// TIA Portal V19 export
FUNCTION_BLOCK "Robot_Modbus"   // FB1, LAD
{ S7_Optimized_Access := 'TRUE' }
// V.0.1.1 - Updated UR robot array address
// V.0.1.0 - Created function block
// stored: MemoryReserve 100, SetENOAutomatically false
   VAR_INPUT
      Proces_Item : Bool;
      Place_Item_Conveyor : Bool;
      Place_Item_Storage : Bool;
      Scrap_Item : Bool;
      Speed_Transport : Int := 10;
      Speed_Grinding : Int := 10;
      Grinding_Coordinates : Bool;
      HMI_String : String;
   END_VAR
   VAR_OUTPUT
      Working : Bool;
      Done : Bool;
      Error : Bool;
      Reached_Coordinates : Bool;
   END_VAR
   VAR
      DISCONNECT : Bool;
      Address : TCON_IP_v4;
      Receive_Data : Int;
      Send_Data : Array[0..63] of Bool;
      Send_Coordinates : Array[0..2] of Int;
      Letter_A : Array[0..20] of "XYZ_Coordinates";
      Letter_Steps { S7_SetPoint := 'True'} : Int;
      Rising_edge : Bool;
      String_To_Letter_Array : Array[0..16] of Char;
      String_Length : Int;
      Currently_Processing : Int;
      Send_Letter_A : Bool;
      Send_Letter_B : Bool;
      Send_Letter_C : Bool;
      MB_Client_Mode : Int;
      MB_Client_Modbus_Address : Int;
      For_Loop_Counter : Int;
   END_VAR
   // Address.InterfaceId := 64;
   // Address.ID := 1;
   // Address.ConnectionType := 11;
   // Address.ActiveEstablished := TRUE;
   // Address.RemoteAddress.ADDR[1] := 192;
   // Address.RemoteAddress.ADDR[2] := 168;
   // Address.RemoteAddress.ADDR[3] := 1;
   // Address.RemoteAddress.ADDR[4] := 51;
   // Address.RemotePort := 502;
   // Address.LocalPort := 502;
   // Letter_A[0..1].X := 4;
   // Letter_A[2].X := 42;
   // Letter_A[3].X := 56;
   // Letter_A[4].X := 98;
   // Letter_A[5].X := 82;
   // Letter_A[6].X := 70;
   // Letter_A[7].X := 29;
   // Letter_A[8].X := 17;
   // Letter_A[9..10].X := 4;
   // Letter_A[11..12].X := 67;
   // Letter_A[13].X := 56;
   // Letter_A[14].X := 52;
   // Letter_A[15].X := 49;
   // Letter_A[16].X := 47;
   // Letter_A[17].X := 44;
   // Letter_A[18..19].X := 33;
   // Letter_A[0].Y := 0;
   // Letter_A[2..3].Y := 100;
   // Letter_A[4..5].Y := 0;
   // Letter_A[6..7].Y := 30;
   // Letter_A[8..10].Y := 0;
   // Letter_A[11..12].Y := 41;
   // Letter_A[13].Y := 69;
   // Letter_A[14].Y := 82;
   // Letter_A[15].Y := 90;
   // Letter_A[16].Y := 80;
   // Letter_A[17].Y := 70;
   // Letter_A[18..19].Y := 41;
   // Letter_A[1..9].Z := -1;
   // Letter_A[10].Z := 0;
   // Letter_A[12..18].Z := -1;
   // Letter_A[19].Z := 0;
   // Letter_A[14].I := 394;
   // Letter_A[15].I := 156;
   // Letter_A[16].I := -122;
   // Letter_A[17].I := -127;
   // Letter_A[14].J := 149;
   // Letter_A[15].J := 53;
   // Letter_A[16].J := 24;
   // Letter_A[17].J := 36;
   VAR_TEMP   // added for the SCL form of the ladder/FBD networks
      _w1 : Bool;
   END_VAR
BEGIN

REGION Network 1: MB_CLIENT
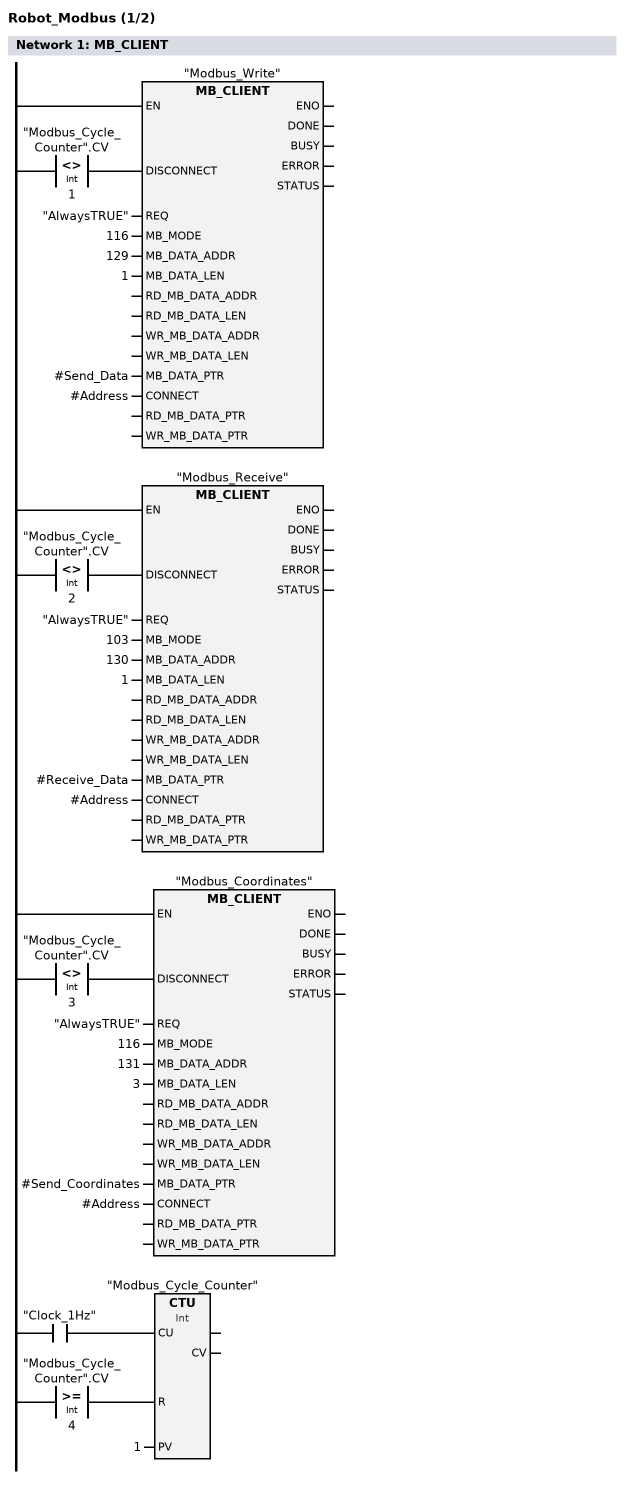
   RUNG wire#powerrail
      "Modbus_Write".MB_CLIENT(DISCONNECT := wire#w1, REQ := "AlwaysTRUE", MB_MODE := 116, MB_DATA_ADDR := 129, MB_DATA_LEN := 1, RD_MB_DATA_ADDR :=, RD_MB_DATA_LEN :=, WR_MB_DATA_ADDR :=, WR_MB_DATA_LEN :=, MB_DATA_PTR := #Send_Data, CONNECT := #Address, RD_MB_DATA_PTR :=, WR_MB_DATA_PTR :=, DONE =>, BUSY =>, ERROR =>, STATUS =>)
   END_RUNG
   RUNG wire#powerrail
      { S7_Templates := "SrcType := Int" } NE_Contact(in1 := "Modbus_Cycle_Counter".CV, in2 := 1)
   END_RUNG wire#w1
   RUNG wire#powerrail
      "Modbus_Receive".MB_CLIENT(DISCONNECT := wire#w2, REQ := "AlwaysTRUE", MB_MODE := 103, MB_DATA_ADDR := 130, MB_DATA_LEN := 1, RD_MB_DATA_ADDR :=, RD_MB_DATA_LEN :=, WR_MB_DATA_ADDR :=, WR_MB_DATA_LEN :=, MB_DATA_PTR := #Receive_Data, CONNECT := #Address, RD_MB_DATA_PTR :=, WR_MB_DATA_PTR :=, DONE =>, BUSY =>, ERROR =>, STATUS =>)
   END_RUNG
   RUNG wire#powerrail
      { S7_Templates := "SrcType := Int" } NE_Contact(in1 := "Modbus_Cycle_Counter".CV, in2 := 2)
   END_RUNG wire#w2
   RUNG wire#powerrail
      "Modbus_Coordinates".MB_CLIENT(DISCONNECT := wire#w3, REQ := "AlwaysTRUE", MB_MODE := 116, MB_DATA_ADDR := 131, MB_DATA_LEN := 3, RD_MB_DATA_ADDR :=, RD_MB_DATA_LEN :=, WR_MB_DATA_ADDR :=, WR_MB_DATA_LEN :=, MB_DATA_PTR := #Send_Coordinates, CONNECT := #Address, RD_MB_DATA_PTR :=, WR_MB_DATA_PTR :=, DONE =>, BUSY =>, ERROR =>, STATUS =>)
   END_RUNG
   RUNG wire#powerrail
      { S7_Templates := "SrcType := Int" } NE_Contact(in1 := "Modbus_Cycle_Counter".CV, in2 := 3)
   END_RUNG wire#w3
   RUNG wire#powerrail
      Contact( "Clock_1Hz" )
      { S7_Templates := "value_type := Int" } "Modbus_Cycle_Counter".CTU(r := wire#w4, pv := 1, cv =>)
   END_RUNG
   RUNG wire#powerrail
      { S7_Templates := "SrcType := Int" } GE_Contact(in1 := "Modbus_Cycle_Counter".CV, in2 := 4)
   END_RUNG wire#w4
   // the same network as SCL:
   "Modbus_Write"(DISCONNECT := "Modbus_Cycle_Counter".CV <> 1,   // MB_CLIENT
                  REQ := "AlwaysTRUE",
                  MB_MODE := 116,
                  MB_DATA_ADDR := 129,
                  MB_DATA_LEN := 1,
                  MB_DATA_PTR := #Send_Data,
                  CONNECT := #Address);
   "Modbus_Receive"(DISCONNECT := "Modbus_Cycle_Counter".CV <> 2,   // MB_CLIENT
                    REQ := "AlwaysTRUE",
                    MB_MODE := 103,
                    MB_DATA_ADDR := 130,
                    MB_DATA_LEN := 1,
                    MB_DATA_PTR := #Receive_Data,
                    CONNECT := #Address);
   "Modbus_Coordinates"(DISCONNECT := "Modbus_Cycle_Counter".CV <> 3,   // MB_CLIENT
                        REQ := "AlwaysTRUE",
                        MB_MODE := 116,
                        MB_DATA_ADDR := 131,
                        MB_DATA_LEN := 3,
                        MB_DATA_PTR := #Send_Coordinates,
                        CONNECT := #Address);
   "Modbus_Cycle_Counter".CTU(CU := "Clock_1Hz", R := "Modbus_Cycle_Counter".CV >= 4, PV := 1);
END_REGION

REGION Network 2: Send Data
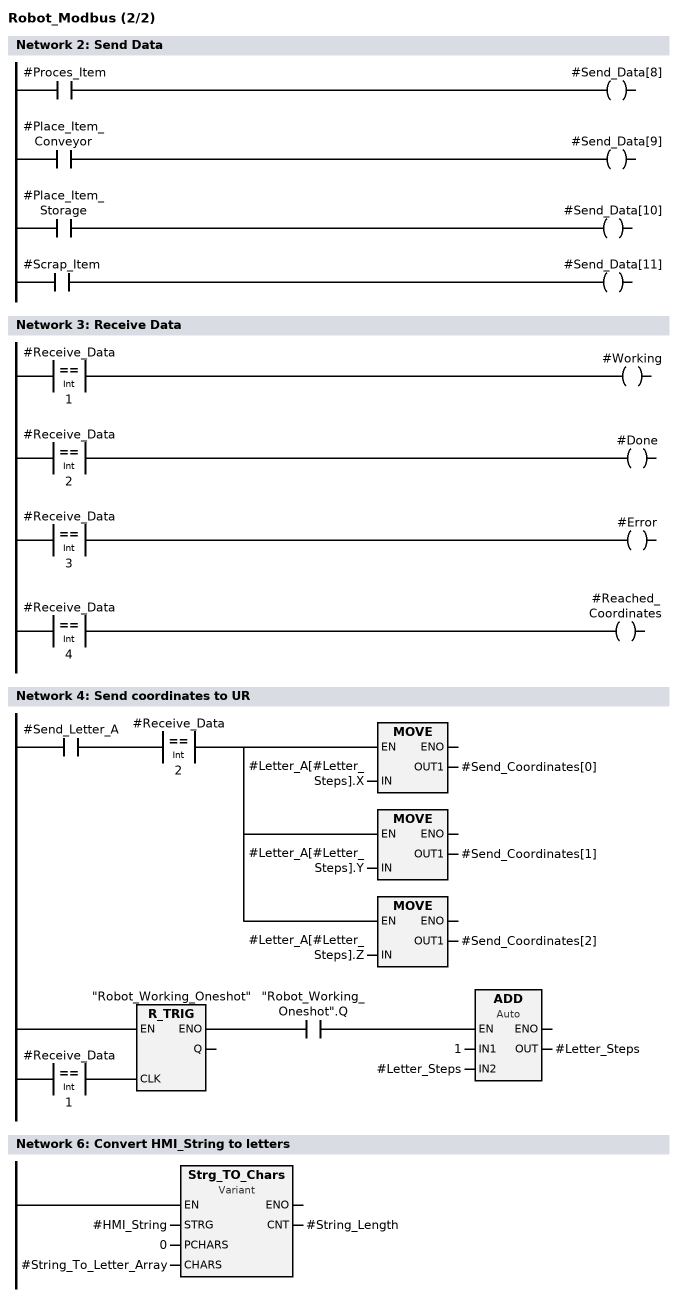
   RUNG wire#powerrail
      Contact( #Proces_Item )
      Coil( #Send_Data[8] )
   END_RUNG
   RUNG wire#powerrail
      Contact( #Place_Item_Conveyor )
      Coil( #Send_Data[9] )
   END_RUNG
   RUNG wire#powerrail
      Contact( #Place_Item_Storage )
      Coil( #Send_Data[10] )
   END_RUNG
   RUNG wire#powerrail
      Contact( #Scrap_Item )
      Coil( #Send_Data[11] )
   END_RUNG
   // the same network as SCL:
   #Send_Data[8] := #Proces_Item;
   #Send_Data[9] := #Place_Item_Conveyor;
   #Send_Data[10] := #Place_Item_Storage;
   #Send_Data[11] := #Scrap_Item;
END_REGION

REGION Network 3: Receive Data
   RUNG wire#powerrail
      { S7_Templates := "SrcType := Int" } EQ_Contact(in1 := #Receive_Data, in2 := 1)
      Coil( #Working )
   END_RUNG
   RUNG wire#powerrail
      { S7_Templates := "SrcType := Int" } EQ_Contact(in1 := #Receive_Data, in2 := 2)
      Coil( #Done )
   END_RUNG
   RUNG wire#powerrail
      { S7_Templates := "SrcType := Int" } EQ_Contact(in1 := #Receive_Data, in2 := 3)
      Coil( #Error )
   END_RUNG
   RUNG wire#powerrail
      { S7_Templates := "SrcType := Int" } EQ_Contact(in1 := #Receive_Data, in2 := 4)
      Coil( #Reached_Coordinates )
   END_RUNG
   // the same network as SCL:
   #Working := #Receive_Data = 1;
   #Done := #Receive_Data = 2;
   #Error := #Receive_Data = 3;
   #Reached_Coordinates := #Receive_Data = 4;
END_REGION

REGION Network 4: Send coordinates to UR
   RUNG wire#powerrail
      Contact( #Send_Letter_A )
      { S7_Templates := "SrcType := Int" } EQ_Contact(in1 := #Receive_Data, in2 := 2)
      wire#w1
      Move(in := #Letter_A[#Letter_Steps].X, out1 => #Send_Coordinates[0])
   END_RUNG
   RUNG wire#w1
      Move(in := #Letter_A[#Letter_Steps].Y, out1 => #Send_Coordinates[1])
   END_RUNG
   RUNG wire#w1
      Move(in := #Letter_A[#Letter_Steps].Z, out1 => #Send_Coordinates[2])
   END_RUNG
   RUNG wire#powerrail
      "Robot_Working_Oneshot".R_TRIG(CLK := wire#w2, Q =>)
      Contact( "Robot_Working_Oneshot".Q )
      Add(in1 := 1, in2 := #Letter_Steps, out => #Letter_Steps)
   END_RUNG
   RUNG wire#powerrail
      { S7_Templates := "SrcType := Int" } EQ_Contact(in1 := #Receive_Data, in2 := 1)
   END_RUNG wire#w2
   // the same network as SCL:
   IF #Send_Letter_A AND (#Receive_Data = 2) THEN
       #Send_Coordinates[0] := #Letter_A[#Letter_Steps].X;
       #Send_Coordinates[1] := #Letter_A[#Letter_Steps].Y;
       #Send_Coordinates[2] := #Letter_A[#Letter_Steps].Z;
   END_IF;
   "Robot_Working_Oneshot"(CLK := #Receive_Data = 1, ENO => #_w1);   // R_TRIG
   IF #_w1 AND "Robot_Working_Oneshot".Q THEN #Letter_Steps := 1 + #Letter_Steps; END_IF;
END_REGION

REGION Network 5 (SCL): Insert coordinates into Modbus_Data array
   (*
   //If we need to make letter A, and robot is sending ready signal
   IF #Send_Letter_A AND #Send_Data[25] THEN

       FOR #For_Loop_Counter := 32 TO 48 DO
           //Find the bit state inside to INT of letter_A array, and copy that to the Modbus data array
           //The for loop repeats the steps again for the array posistions 32-48
           #Letter_A[#Letter_Steps].X.%X0 := #Send_Data[#For_Loop_Counter];
       END_FOR;

       FOR #For_Loop_Counter := 49 TO 64 DO
           #Letter_A[#Letter_Steps].Y.%X0 := #Send_Data[#For_Loop_Counter];
       END_FOR;

       FOR #For_Loop_Counter := 65 TO 79 DO
           #Letter_A[#Letter_Steps].Z.%X0 := #Send_Data[#For_Loop_Counter];
       END_FOR;

   END_IF; *)
END_REGION

REGION Network 6: Convert HMI_String to letters
   RUNG wire#powerrail
      { S7_Templates := "[ptr_type := Variant, strg_type := String]" } Strg_TO_Chars(Strg := #HMI_String, pChars := 0, Chars := #String_To_Letter_Array, Cnt => #String_Length)
   END_RUNG
   // the same network as SCL:
   Strg_TO_Chars(Strg := #HMI_String, pChars := 0, Chars := #String_To_Letter_Array, Cnt => #String_Length);
END_REGION

REGION Network 7 (SCL)
   IF #Currently_Processing < #String_Length THEN //Hvis vi ikke er nået forbi enden af teksten

       IF #String_To_Letter_Array[#Currently_Processing] = 'A' THEN //Hvis der på position X, er et "A" i teksten
           #Send_Letter_A := TRUE;
       ELSIF #String_To_Letter_Array[#Currently_Processing] = 'B' THEN
           #Send_Letter_B := TRUE;
       ELSIF #String_To_Letter_Array[#Currently_Processing] = 'C' THEN
           #Send_Letter_B := TRUE;
       END_IF;
   END_IF;
END_REGION
END_FUNCTION_BLOCK
